FUNCTION_BLOCK randnum
VAR_OUTPUT
    RandomNumber : LREAL; (* Generated random number *)
END_VAR

VAR
    DRANDFB : DRAND; (* Function Block instance for generating random numbers *)
	MinValue : LREAL := 10.0; (* Minimum value of the range *)
    MaxValue : LREAL := 50.0; (* Maximum value of the range *)
END_VAR

(* Generate a random number and scale it to the desired range *)
DRANDFB(Seed := 1); (* Call to generate a random number *)
RandomNumber := MinValue + (MaxValue - MinValue) * DRANDFB.Num;

END_FUNCTION_BLOCK

(* stored: Version 1.1.0.1
   POU randnum: Id {207dc5b8-8440-4437-9179-542f78bfc425}, SpecialFunc None *)
